{attribute 'enable_dynamic_creation'}
FUNCTION_BLOCK RecipeSingleValue IMPLEMENTS RecipeSingleValueType
VAR
	_Name : T_MaxString;
	_Value : __SYSTEM.AnyType;
	_Assignment : STRING := ':=';
	_AssignmentString : T_MaxString;
END_VAR

{attribute 'monitoring' := 'call'}
PROPERTY Assignment : STRING
GET
Assignment := _Assignment;
END_GET
SET
_Assignment := Assignment;
END_SET
END_PROPERTY

METHOD Bind
VAR_INPUT
	value : ANY;
END_VAR
_Value := value;
END_METHOD

METHOD BuildAndGetAssignmentString : POINTER TO STRING
VAR_INPUT
END_VAR
_AssignmentString := 
	BuildStringInline(_Name)
	.Append(_Assignment)
	.Append(ValueString)
	.GetString();
BuildAndGetAssignmentString := ADR(_AssignmentString);
END_METHOD

METHOD Dispose
VAR_INPUT
END_VAR
__DELETE(THIS);
END_METHOD

{attribute 'monitoring' := 'call'}
PROPERTY Name : T_MaxString
GET
Name := _Name;
END_GET
SET
_Name := Name;
END_SET
END_PROPERTY

METHOD ParseAndAssignValue
VAR_INPUT
	value : T_MaxString;
END_VAR
StringToAnyType(value, _Value);
END_METHOD

{attribute 'monitoring' := 'call'}
PROPERTY ValueString : T_MaxString
GET
IF (IsAnyTypeBound(_Value)) THEN
	ValueString := AnyTypeToString(_Value);
END_IF
END_GET
END_PROPERTY

END_FUNCTION_BLOCK

(* stored: Version 1.1.0.1
   POU RecipeSingleValue: Id {942ad2e3-e169-0d10-23b7-39164624dfb7}, SpecialFunc None
   Property Assignment: Id {f2e379a6-6acc-0cb4-3f61-526d7942b9e8}
   Get Get: Id {803a6e83-74e6-0f1e-00a3-e65750706004}
   Set Set: Id {3ddf8cbe-8880-015e-2b54-049636be31d7}
   Method Bind: Id {53f3350b-066f-0459-2828-74755586ae97}
   Method BuildAndGetAssignmentString: Id {f950f745-9204-0d83-0156-682978ab7e06}
   Method Dispose: Id {20effca3-ad4b-0592-28db-63b359f9939a}
   Property Name: Id {f5f59799-4de8-0350-1461-82001d0fab6e}
   Get Get: Id {2277b73e-3ebe-0763-348b-5c19875b9a80}
   Set Set: Id {d054d088-4dc5-003f-34b6-72da849ecf8e}
   Method ParseAndAssignValue: Id {ba3fab94-a61b-0cea-03fa-c1d2fb0eef56}
   Property ValueString: Id {e677d293-dd1f-0c68-237c-9798e0861df8}
   Get Get: Id {1735fe82-6618-0f32-1e2b-d212e7d4fb07} *)
